TYPE ST_MonitoredAttribute :
STRUCT
	attribute : FB_MonitoredAttribute;
	attributeId : DINT;
	deviceId : DINT;
END_STRUCT
END_TYPE

(* stored: Version 1.1.0.1, ProductVersion 3.1.4024.12
   DUT ST_MonitoredAttribute: Id {e11813d7-723a-44d8-b978-76d793f1a6ea} *)
